{attribute 'linkalways'} 
{attribute 'no_explicit_call' := 'This FB is a CLASS and must be accessed using methods or properties'}
{attribute 'enable_dynamic_creation'}
FUNCTION_BLOCK FINAL LT_LWORD EXTENDS Node
VAR
	in1 : _LWORD(0);
	in2 : _LWORD(0);
	out : _BOOL(FALSE);
END_VAR

METHOD PUBLIC Clone : I_Node
VAR
	pNode : POINTER TO LT_LWORD;
END_VAR
pNode := __NEW(LT_LWORD);
Clone := pNode^;
END_METHOD

METHOD FB_init : BOOL
VAR_INPUT
	bInitRetains : BOOL; // if TRUE, the retain variables are initialized (warm start / cold start)
	bInCopyCode : BOOL;  // if TRUE, the instance afterwards gets moved into the copy code (online change)
END_VAR
AddInput('in1',THIS^.in1);
AddInput('in2',THIS^.in2);
AddOutput('out', THIS^.out);
END_METHOD

METHOD PROTECTED OnExecute
VAR
END_VAR
out.Value := in1.Value < in2.Value;
END_METHOD

END_FUNCTION_BLOCK

(* stored: Version 1.1.0.1, ProductVersion 3.1.4024.15
   POU LT_LWORD: Id {b9b045a1-c8d8-4d32-91e7-90d8bf3a1ff1}, SpecialFunc None
   Folder Constructor: Id {6e87b6c0-bf28-4c74-9a00-c681e91409b6}
   Method Clone: Id {40fa957f-210b-4f85-a6da-cff667b7c8c3}
   Method FB_init: Id {c3eccfd5-ef9a-4e83-b685-67f359290c1c}
   Method OnExecute: Id {0217f3eb-30c2-48a2-9391-4088a6f405b5} *)
